PROGRAM AzimuthElevationControl
VAR_INPUT
	// decrease azimuth
	left:		BOOL;
	// increase azimuth
	right: 		BOOL;
	// reset the axis
	Reset: 		BOOL;
	// enable the axis and its position control loop
	Enable:		BOOL;
	// Move azimuth to given position
	MoveAxis:	BOOL;
	// Home the axis
	HomeAxis:	BOOL;
	// enable tracking
	Tracking:	BOOL;
	// position to move the axis to
	position: 	LREAL;
END_VAR
VAR_OUTPUT
	// error state of the axis
	error: 			BOOL;
	// error ID of the axis
	ErrorID:		UDINT;
	// actual_position of the axis
	act_position:	LREAL;
	// is the axis calibrated
	calibrated:		BOOL;
	// drive is ready
	ready:			BOOL;
	// time to reach target position
	slewtime:		LREAL;
END_VAR
VAR
	AzimuthAxis:		FB_Axis2;
	AzimuthCalibration: MC_SetPosition;
	fbSoEReset:			FB_SoEReset;
	AzimuthAxisEvent: 	FB_EventLog;
	// delay until commutator angle is measured
	readydelay:			TON;
	HomeDelay:			FB_TONTP;
	TorqueError:		TON := (PT := T#3S);
	azimuth_torque: 	REAL;
	TorqueWarning:		FB_EventLog;
	CalibrationEvent:	FB_Eventlog;
	ReadParameter:		MC_ReadParameter;
	getlastposition:	BOOL := TRUE;
	bSoEReset:			BOOL;
END_VAR
VAR CONSTANT
	// reference position for homing
	// homing_position:		LREAL := 439.0; // was 442 - -21.21 = 463.21; 463 + 24 = 439
	// current position of the calibration cam encoder zero index. Apply an offset here if necessary
	calibration_position:	LREAL := 156.1195; // 393.0; 
END_VAR
VAR PERSISTENT
	last_position:	LREAL := -1.0;
END_VAR

(* Azimuth Axis control section
Power must be on and brake must be open for the axis to operate
*)

// generate the ready signal after enabling the drive
readydelay(IN :=  AzimuthAxis.Enable, PT := T#3000MS, Q=> ready);

// limit the input position angle
position := LIMIT(0.0, position, 450.0);

// conduct the calibrated signal
calibrated := AzimuthAxis.Calibrated;

IF Calibrated OR Error THEN
	HomeAxis := FALSE;
	getlastposition := FALSE;
END_IF
	
IF HomeAxis THEN
	position := calibration_position;
END_IF

(*
// move to calibration_position after homing
HomeDelay(IN := Calibrated, PT1 := T#5S, PT2 := T#100MS);
*)
IF HomeDelay.Q THEN
	position := calibration_position;
	MoveAxis := TRUE;
END_IF

// perform a recalibration on the last known position
AzimuthCalibration(
	Axis := GVL_Telescope.AzimuthAxisRef,
	Execute := getlastposition AND last_position>=0.0 AND NOT Calibrated,
	Position := last_position);

IF AzimuthCalibration.Done THEN
	getlastposition := FALSE;
END_IF

IF Calibrated THEN
	last_position := act_position;
END_IF
	
// deactivate limit switches on homing
MC_SetAcceptBlockedDriveSignal(
	Axis := GVL_Telescope.AzimuthAxisRef, 
	Enable := HomeAxis);

AzimuthAxis(	
	Enable := 			enable AND HydraulicsControl.brake_open AND HydraulicsControl.oil_pressure_OK,
	Reset := 			reset,
	MoveAxis :=			MoveAxis,
	HomeAxis := 		HomeAxis,
	Tracking :=			Tracking,
	Position := 		position, 
	Enable_Positive := 	NOT GVL_Telescope.azimut_limit_switch AND (GVL_Telescope.Azimuth_inputs.1 OR HomeAxis),
	Enable_Negative := 	NOT GVL_Telescope.azimut_limit_switch AND GVL_Telescope.Azimuth_inputs.0,
	Jog_Forward :=		right,
	Jog_Backwards := 	left,
	bCalibrationCam :=	NOT GVL_Telescope.Azimuth_inputs.1,
	ActualPosition => 	act_position,
	Error => 			error,
	ErrorID => 			ErrorID,
	AxisRef :=			GVL_Telescope.AzimuthAxisRef);

bSoEReset := GVL_Telescope.Azimuth_diagnostic = 16#0000F10B OR GVL_Telescope.Azimuth_diagnostic = 16#0000F601;

IF bSoEReset THEN
	last_position := -1.0;
	fbSoEReset(
		Axis := GVL_Telescope.AzimuthAxisRef,
		Execute := TRUE,
		Timeout := DEFAULT_ADS_TIMEOUT);
 	IF fbSoEReset.Busy THEN
		fbSoEReset(Axis := GVL_Telescope.AzimuthAxisRef, Execute := FALSE);
	ELSE
		bSoEReset := FALSE;
		Reset := TRUE;
	END_IF
END_IF 
	
IF AzimuthAxis.MoveDone THEN
	MoveAxis := FALSE;
END_IF

IF AzimuthAxis.HomeDone THEN
	HomeAxis := FALSE;
END_IF
	
IF AzimuthAxis.ResetDone THEN
	reset := FALSE;
END_IF

ReadParameter(	Axis := GVL_Telescope.AzimuthAxisRef, Enable := AzimuthAxis.InMotion, 
				ParameterNumber := MC_AxisParameter.AxisRemainingTimeToGo, 
				ReadMode := E_ReadMode.READMODE_CYCLIC);
IF ReadParameter.Valid THEN
	slewtime := ReadParameter.Value;
END_IF

azimuth_torque := GVL_Telescope.Azimuth_torque / 10.0;
TorqueError(IN := ABS(azimuth_torque) > 50.0);


AzimuthAxisEvent(	
	Trigger := 		Error, 
	Level := 		ADSLOG_MSGTYPE_ERROR,
	FormatString :=	'Azimuth Axis Error: %s',
	OnMessage := 	NCError_TO_STRING(ErrorID));
	
TorqueWarning(	
	Trigger := 		TorqueError.Q, 
	Level := 		ADSLOG_MSGTYPE_WARN,
	FormatString :=	'%s',
	OnMessage := 	'Azimuth torque is high.');
	
CalibrationEvent(
	Trigger := 		Calibrated, 
	Level := 		ADSLOG_MSGTYPE_HINT,
	FormatString :=	'%s',
	OnMessage := 	'Azimuth axis is calibrated.');

END_PROGRAM

(* stored: Version 1.1.0.1, ProductVersion 3.1.4024.9
   POU AzimuthElevationControl: Id {8e08648a-b748-4448-9dcc-aa13dfcf6a06}, SpecialFunc None *)
